# EPICS substitutions: bkpApp/Db/bkp.substitutions
file bkpCommon.template {
pattern
{None}
{None}
}

#file bkpCh.template {
#pattern
#{CHAN}
#{   1}
#{   2}
#{   3}
#}
